FUNCTION_BLOCK Transportwagen
VAR_INPUT
END_VAR
VAR_OUTPUT
END_VAR
VAR
END_VAR

SimDA.P1:= SimDI.S1;
SimDA.Q1:= SimDI.S2;
SimDA.Q2:= SimDI.S3;

END_FUNCTION_BLOCK

(* stored: Version 1.1.0.1, ProductVersion 3.1.4024.5
   POU Transportwagen: Id {f156885e-d892-4706-970d-8d2a74171c01}, SpecialFunc None *)
